# EPICS autosave request: calc/calcApp/Db/interpNew_settings.req
$(P)interp$(Q)_mode
$(P)interp$(Q).VALA
$(P)interp$(Q).VALB
$(P)interp$(Q).VALC
$(P)interp$(Q).VALN
$(P)interp$(Q).F
$(P)interp$(Q)_n
$(P)interp$(Q)_x
$(P)interp$(Q)_y1
$(P)interp$(Q)_y1.OUT
$(P)interp$(Q)_y1.DESC
$(P)interp$(Q)_y2
$(P)interp$(Q)_y2.OUT
$(P)interp$(Q)_y2.DESC
